FUNCTION Simulatie_invoer : BOOL
VAR_INPUT
END_VAR
VAR
	timer1: TON;
END_VAR



IF GVL.ZaagLengte <= GVL.HuidigePositieAanvoer THEN
	Gvl.MotorInvoer:= TRUE;				
	GVL.HuidigePositieAanvoer := GVL.HuidigePositieAanvoer - 1;
END_IF;
			
			
IF GVL.ZaagLengte > GVL.HuidigePositieAanvoer THEN
	Gvl.MotorInvoer:= TRUE;				
	GVL.HuidigePositieAanvoer := GVL.HuidigePositieAanvoer + 1;
END_IF;


IF GVL.ZaagLengte = GVL.HuidigePositieAanvoer THEN
GVL.MotorInvoer := FALSE;
END_IF

END_FUNCTION

(* stored: Version 1.1.0.1, ProductVersion 3.1.4024.12
   POU Simulatie_invoer: Id {371512e1-b4c3-4157-99ae-e3d8e8edb7d8}, SpecialFunc None *)
